PROGRAM PRG_OPT
VAR
	bInit: BOOL := TRUE;
	fbMotionRxG: FB_MotionStage;
	fbMotionXG: FB_MotionStage;
	fbMotionRzPM: FB_MotionStage;
END_VAR

IF bINIT THEN
	
	GVL_Main.M10.nBrakeMode := ENUM_StageBrakeMode.NO_BRAKE;
	GVL_Main.M10.bHardwareEnable := TRUE;
	GVL_Main.M10.bPowerSelf := TRUE;
	GVL_Main.M11.nBrakeMode := ENUM_StageBrakeMode.NO_BRAKE;
	GVL_Main.M11.bHardwareEnable := TRUE;
	GVL_Main.M11.bPowerSelf := TRUE;
	GVL_Main.M14.nBrakeMode := ENUM_StageBrakeMode.NO_BRAKE;
	GVL_Main.M14.bHardwareEnable := TRUE;
	GVL_Main.M14.bPowerSelf := TRUE;

	bINIT := FALSE;
END_IF;


fbMotionRxG(stMotionStage:= GVL_Main.M10);
fbMotionXG(stMotionStage:= GVL_Main.M11);
fbMotionRzPM(stMotionStage:= GVL_Main.M14);

END_PROGRAM

(* stored: Version 1.1.0.1, ProductVersion 3.1.4022.18
   POU PRG_OPT: Id {9fd4ef96-d0b3-4d92-a155-89dc0eb4c6d2}, SpecialFunc None *)
